{attribute 'GeneratedUsingTerminal: EK1122-0000-0018'}
{attribute addProperty BoxType "EK1122-0000-0018"}
{attribute addProperty Id "Beckhoff_EL68xxsub_EK1100EK1100_1FC0878B2"}
{attribute addProperty CRC "2753407709"}
{attribute addProperty Size "2"}
TYPE Beckhoff_EL68xxEK1122_A41DAADD EXTENDS EK1122_1FC0878B :
STRUCT
	{attribute addProperty Name "Beckhoff EL68xxsub EK1100"}
	{attribute addProperty PreviousPort "Beckhoff EL68xxEK1122 : D"}
	Beckhoff_EL68xxsub_EK1100 : EK1100_1FC0878B;
END_STRUCT
END_TYPE

(* stored: Version 1.2.0.0, ProductVersion 3.1.4024.9
   DUT Beckhoff_EL68xxEK1122_A41DAADD: Id {e217369d-b40c-4f4b-8387-b3af9fa68b6b} *)
